(* CoDeSys 2.3 export: BR_REQ.EXP *)

(* Data type *)
TYPE BR_REQ :
	(
	BR_NONE_REQ := 0,
	BR_SINS1_REQ,
	BR_SINS2_REQ,
	BR_SINS3_REQ,
	BR_YAG_REQ
	);
END_TYPE
